TYPE ST_ErrorDataSet :
(**************************************************************************************
 * 	Application		:	BoxControl Framework
 *	Revision		:	$Revision: 404529 $
 *	Revision date	:	$Date: 2018-04-23 08:21:38 +0200 (Mo., 23 Apr 2018) $
 *	Last changed by	:	$Author: b7bolm $
 *	URL				:	$URL: http://almscdc.swisslog.com/repo/SWPD/Development/BoxControlFramework/20_Release/trunk/01_Software/BCF/BCF/JumpStart/20_Product/10_App/10_Base/10_Lib/10_Conv/01_DUTs/ST_ErrorDataSet.TcDUT $
 *
 *	Purpose			:	Error data set
 *
 * ------------------------------------------------------------------------------------
 *	Copyright Swisslog [IP AG], Switzerland. All rights reserved.
 * 
 * ------------------------------------------------------------------------------------
 *	
 * 	Revision History: 
 *
 * 	VERSION			DATE			INITIALS			DESCRIPTION
 *	0.1				01.01.2001		swl					Example
 *
 **************************************************************************************)
STRUCT
	ErrorType		: E_ErrorType;	// Type of error 
	ErrorCode		: U_ErrorCode; // Type casting for error code by product or framework errors 
	ErrorParam		: STRING(System.ERROR_PARAM_STRINGLENGTH); // Error parameter 
	ResetError		: BOOL; // Command to reset error 
END_STRUCT
END_TYPE

(* stored: Version 1.1.0.1, ProductVersion 3.1.4022.12
   DUT ST_ErrorDataSet: Id {c0cb4f30-d0c5-44ff-a8ff-5d960d53c8c1} *)
